RoboDK station: PP.rdk

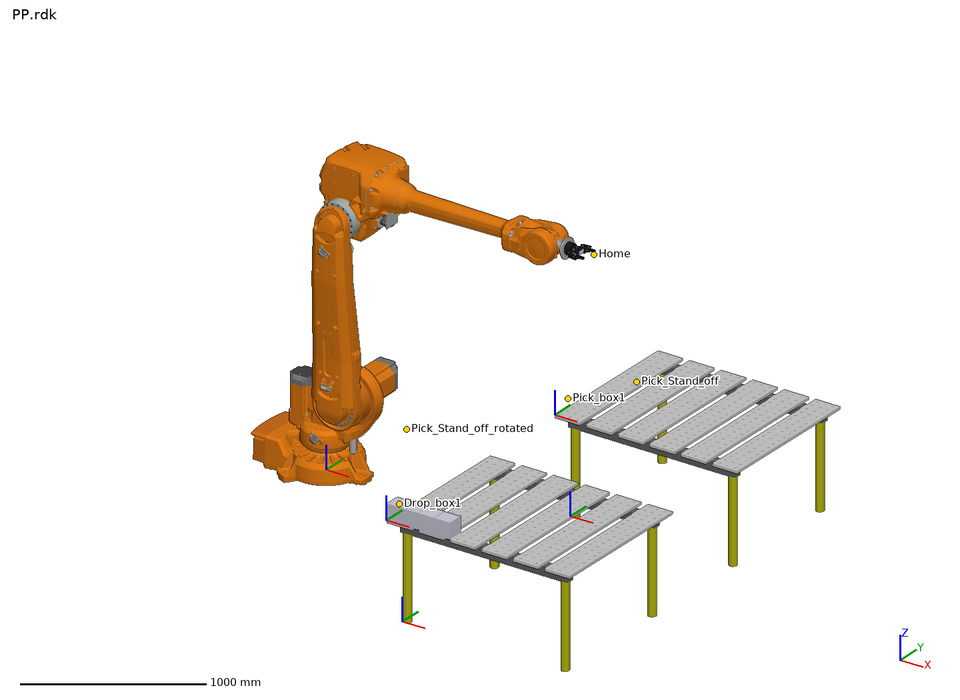
[picture v0: the station drawn from its stored meshes, robots at their saved joint values, targets as dots, program paths as lines]
Station New Station (1) (saved by RoboDK 5.1.2). Poses are relative to the parent item; angles as X-Y-Z fixed-axis rotations.
  - frame ABB IRB 4600-40/2.55 Base at (578.84, -764, 0) mm
    - robot ABB IRB 4600-40/2.55: 6 axes, payload 40 kg, reach 2550 mm, repeatability 0.06 mm, weight 435 kg
        modified DH rows (alpha deg, a mm, theta deg, d mm): 0, 0, 0, 495; -90, 175, -90, 0; 0, 1095, 0, 0; -90, 175, 0, 1270; 90, 0, 0, 0; -90, 0, 180, 135
        joint limits [-180, -90, -180, -400, -125, -400] to [180, 150, 75, 400, 120, 400]; home [0, 0, 0, 0, 0, 0]; saved at [0, 0, 0, 0, 0, 0]
      - tool Tool, TCP at (0, 0, 130) mm, size 147.4 x 146.8 x 75 mm
    - target Pick_Stand_off (joint target) at (2033.58, 0, 1091.98) mm, rotated rx 180 ry 3.2 rz 180 deg; joints [0, 30.11, -20.37, 0, 77.06, 0] of ABB IRB 4600-40/2.55
    - target Home (joint target) at (1753.96, 0, 1775.72) mm, rotated rx 0 ry 90 rz 0 deg; joints [0, 0, 0, 0, 0, 0] of ABB IRB 4600-40/2.55
    - target Pick_Stand_off_rotated (joint target) at (674.22, -212.99, 516.32) mm, rotated rx 176.8 ry 0 rz 90 deg; joints [0, 30.11, -20.37, 0, 77.06, 90] of ABB IRB 4600-40/2.55
  - folder Objects
    - frame Table_pick_base at (1987.97, -493.84, 9.53) mm
      - object Table at (533.9, 425.22, 609.31) mm, size 1193.8 x 965.2 x 609.6 mm, geometry from welding_table.sld
    - frame Table_pick_top at (1925.03, -551.01, 618.96) mm
      - target Pick_box1 (joint target) at (50, 50, 90) mm, rotated rx 180 ry 3.2 rz -180 deg; joints [10.779, 5.473, 30.86, -0.775, 50.526, 11.255] of ABB IRB 4600-40/2.55
    - frame Table_drop_base at (1987.97, -2062.15, 9.53) mm
      - object Table at (533.9, 425.22, 609.31) mm, size 1193.8 x 965.2 x 609.6 mm, geometry from welding_table.sld
      - frame Table_drop_top at (-64.7, -59.62, 609.97) mm
        - target Drop_box1 (joint target) at (50, 50, 90) mm, rotated rx -180 ry 3.2 rz 90 deg; joints [-42.838, 29.317, 0.309, -2.76, 58.228, 48.571] of ABB IRB 4600-40/2.55
        - object box1 at (50, 50, 50) mm, rotated rx 0 ry 0 rz -90 deg, size 100 x 100 x 100 mm, geometry from box.sld
        - object box2 at (155, 50, 50) mm, rotated rx 0 ry 0 rz -90 deg, size 100 x 100 x 100 mm, geometry from box.sld
        - object box3 at (260, 50, 50) mm, rotated rx 0 ry 0 rz -90 deg, size 100 x 100 x 100 mm, geometry from box.sld
        - object box4 at (365, 50, 50) mm, rotated rx 0 ry 0 rz -90 deg, size 100 x 100 x 100 mm, geometry from box.sld
  - folder Programs
    - program Gripper_Attach (1 instructions, listed below)
    - program Gripper_Dettach (1 instructions, listed below)
  - Python program PP_PRG (listed below)

--- program Gripper_Attach (robot ABB IRB 4600-40/2.55) ---
  Attach to Gripper RobotiQ 85 Opened

--- program Gripper_Dettach (robot ABB IRB 4600-40/2.55) ---
  Detach from Gripper RobotiQ 85 Opened

--- Python program PP_PRG ---
# Type help("robolink") or help("robodk") for more information
# Press F5 to run the script
# Documentation: https://robodk.com/doc/en/RoboDK-API.html
# Reference:     https://robodk.com/doc/en/PythonAPI/index.html
# Note: It is not required to keep a copy of this file, your python script is saved with the station
from robolink import *    # RoboDK API
from robodk import *      # Robot toolbox
RDK = Robolink()

# Any interaction with RoboDK must be done through
# Robolink()
RL = Robolink()


# get the robot item:
robot = RL.Item('ABB IRB 4600-40/2.55')
robottool = RL.Item('Tool')


# get frames
F_top_pick_table = RL.Item('Table_pick_top')
F_top_drop_table = RL.Item('Table_drop_top')

# get the targets:
P_home = RL.Item('Home')
P_pso = RL.Item('Pick_Stand_off')
P_pso_rotated = RL.Item('Pick_Stand_off_rotated')
P_pb1 = RL.Item('Pick_box1')
P_db1 = RL.Item('Drop_box1')





# move the robot to home, then to Stand off Position:
robot.MoveJ(P_home)
robot.MoveJ(P_pso)


poseref_pick = P_pb1.Pose()

poseref_drop = P_db1.Pose()


for i in range(0,365,105):

    robot.setSpeed(100,100)
    robot.setPoseFrame(F_top_pick_table)

    posei = poseref_pick.Offset(i,0,200)
    robot.MoveJ(posei)
    posei = poseref_pick.Offset(i,0,0)
    robot.MoveL(posei)
    robottool.AttachClosest()
    posei = poseref_pick.Offset(i,0,200)
    robot.MoveL(posei)

    #move the robot to stand off position
    #robot.MoveJ(P_pso)
    robot.MoveJ(P_pso_rotated)

    #move the robot to drop off position box 1
    robot.setPoseFrame(F_top_drop_table)
    posei = poseref_drop.Offset(i,0,200)
    robot.MoveJ(posei)
    posei = poseref_drop.Offset(i,0,0)
    robot.MoveL(posei)
    robottool.DetachAll(F_top_drop_table)
    posei = poseref_drop.Offset(i,0,200)
    robot.MoveL(posei)

    #move the robot to stand off position
    robot.MoveJ(P_pso)




for i in range(315,-105,-105):

    #move the robot to drop off position box 1
    robot.setPoseFrame(F_top_drop_table)
    posei = poseref_drop.Offset(i,0,200)
    robot.MoveJ(posei)
    posei = poseref_drop.Offset(i,0,0)
    robot.MoveL(posei)
    robottool.AttachClosest()
    posei = poseref_drop.Offset(i,0,200)
    robot.MoveL(posei)

    #move the robot to stand off position
    robot.MoveJ(P_pso)


    robot.setPoseFrame(F_top_pick_table)
    posei = poseref_pick.Offset(i,0,200)
    robot.MoveJ(posei)
    posei = poseref_pick.Offset(i,0,0)
    robot.MoveL(posei)
    robottool.DetachAll(F_top_drop_table)
    posei = poseref_pick.Offset(i,0,200)
    robot.MoveL(posei)

    #move the robot to stand off position
    robot.MoveJ(P_pso)


# # move back to the center, then home:

robot.MoveJ(P_home)
